# EPICS substitutions: iocs/oxigrafMO2iIOC/oxigrafMO2iTestApp/Db/MO2i.substitutions
file MO2i.template
{
	pattern
	{  PRIM,   LOCA,       UNIT,      SCAN,        PORT    }
	{ "ODH", "$(LOCA)", "$(UNIT)", ".5 second",  "$(PORT)" }
}
